FUNCTION_BLOCK FB_RobotTCPReceive
VAR_INPUT
	bEnable : BOOL;
	Robot : STRING;
	bRecordData : BOOL;

END_VAR
VAR_OUTPUT
	bBusy : BOOL;
	bConnected : BOOL;
	bError : BOOL;
	
	
END_VAR
VAR
	data : ARRAY [1..1500] OF BYTE;
	packageData : ARRAY [1..500] OF BYTE;
	eState : E_RobotTCPReceive;
	
	fbSocketConnect : FB_SocketConnect := (sSrvNetId := '', tTimeout := DEFAULT_ADS_TIMEOUT);
	fbSocketClose : FB_SocketClose := (sSrvNetId := '', tTimeout := DEFAULT_ADS_TIMEOUT);
	fbSocketReceive : FB_SocketReceive := (sSrvNetId := '', tTimeout := DEFAULT_ADS_TIMEOUT, cbLen := 1500); //1076
	fbParseURData : FB_ParseURData;
	fbRecordData : FB_CSV_RobotDataWriter;
	
	hSocket1: T_HSOCKET;
	bParsingData: BOOL;

END_VAR

// TCP/IP Messaging Case
CASE eState OF
	
	E_RobotTCPReceive.Idle:
		IF bEnable THEN
			bBusy := TRUE;
			IF NOT bConnected THEN
				eState := E_RobotTCPReceive.Connect_Start;
			ELSE
				eState := E_RobotTCPReceive.Receive_Start;
			END_IF
		ELSIF bConnected THEN
			eState := E_RobotTCPReceive.Close_Start;
		END_IF
	
	E_RobotTCPReceive.Connect_Start:
		fbSocketConnect.bExecute := TRUE;
		fbSocketConnect.nRemotePort := 30001;
		IF Robot='UR3' THEN
			fbSocketConnect.sRemoteHost := Global.stUR3.IP;	
		ELSIF Robot='UR5' THEN
			fbSocketConnect.sRemoteHost := Global.stUR5.IP;
		ELSE
			eState := E_RobotTCPReceive.HandleError;
		END_IF
		eState := E_RobotTCPReceive.Connect_Wait;
		
	E_RobotTCPReceive.Connect_Wait:
		fbSocketConnect.bExecute := FALSE;	
		IF fbSocketConnect.bError THEN
			eState := E_RobotTCPReceive.HandleError;
		ELSIF NOT fbSocketConnect.bBusy THEN
			bConnected := TRUE;
			hSocket1 := fbSocketConnect.hSocket;
			eState := E_RobotTCPReceive.Idle;
		END_IF
		
	E_RobotTCPReceive.Receive_Start:
		fbSocketReceive.bExecute := TRUE;
		fbSocketReceive.hSocket := hSocket1;
		fbSocketReceive.pDest := ADR(data);
		eState := E_RobotTCPReceive.Receive_Wait;
	
	E_RobotTCPReceive.Receive_Wait:
		fbSocketReceive.bExecute := FALSE;
		IF fbSocketReceive.bError THEN
			eState := E_RobotTCPReceive.HandleError;
		ELSIF NOT fbSocketReceive.bBusy THEN
			bParsingData := TRUE;
			eState := E_RobotTCPReceive.ParseData;
		END_IF
		
	E_RobotTCPReceive.ParseData:
		IF bParsingData THEN	
			fbParseURData( data := data, Robot:=Robot);  // Parse and Record UR Data
			bParsingData := FALSE;
			//eState := E_RobotTCPReceive.Idle;
		ELSE
			eState := E_RobotTCPReceive.Idle;
		END_IF
		IF bRecordData THEN
			fbRecordData.bEnable := TRUE;
			IF Robot='UR3' THEN
				fbRecordData.sFileName := 'UR3Data';
				fbRecordData.stRobotData := Global.stUR3;
			ELSIF Robot='UR5' THEN
				fbRecordData.sFileName := 'UR5Data';
				fbRecordData.stRobotData := Global.stUR5;
			END_IF

			fbRecordData.bWriteLine := TRUE;
			
			eState := E_RobotTCPReceive.RecordData_Wait;
		ELSE 
			eState := E_RobotTCPReceive.Idle;
			fbRecordData.bEnable := FALSE;
		END_IF
		
	E_RobotTCPReceive.RecordData_Wait:
		IF fbRecordData.bError THEN
			eState := E_RobotTCPReceive.HandleError;
		ELSIF NOT fbRecordData.bBusy THEN
			eState := E_RobotTCPReceive.Idle;
		END_IF
		
	E_RobotTCPReceive.Close_Start:
		fbSocketClose.bExecute := TRUE;
		fbSocketClose.hSocket := hSocket1;
		eState := E_RobotTCPReceive.Close_Wait;
	
	E_RobotTCPReceive.Close_Wait:
		fbSocketClose.bExecute := FALSE;
		IF fbSocketClose.bError THEN
				eState := E_RobotTCPReceive.HandleError;
		ELSIF NOT fbSocketClose.bBusy THEN
			bConnected := FALSE;
			MEMSET(ADR(hSocket1),0,SIZEOF(hSocket1));
			bBusy := FALSE;
			bError := FALSE;
			eState := E_RobotTCPReceive.Idle;
		END_IF
		
	E_RobotTCPReceive.HandleError:
		bError := TRUE;
		IF bConnected THEN
			eState := E_RobotTCPReceive.Close_Start;
		ELSE
			bBusy := FALSE;
			eState := E_RobotTCPReceive.Idle;
		END_IF
		
END_CASE

fbRecordData();
fbSocketConnect();
fbSocketReceive();
fbSocketClose();

END_FUNCTION_BLOCK

(* stored: Version 1.1.0.1, ProductVersion 3.1.4020.12
   POU FB_RobotTCPReceive: Id {8049a8bc-c88a-46b6-885c-8d0914a443b2}, SpecialFunc None *)
